# EPICS substitutions: iocBoot/ioc13idd/SIS3820_8.substitutions
# This loads the scaler record and supporting records
file "$(STD)/stdApp/Db/scaler.db"
{
pattern
{P,           S,          DTYP,           OUT,                     FREQ}
{13IDD:  scaler2,  "Asyn Scaler",  "@asyn(mcaSIS3820/1 0)",    50000000}
}

# This database provides the record for callbacks when acquisition is complete
file "$(MCA)/mcaApp/Db/SIS3820.db"
{
pattern
{P,         INP}
{13IDD:SIS1:  "@asyn(mcaSIS3820/1 0)"}
}

# This database provides the logic for multiple mca records
file "$(MCA)/mcaApp/Db/Struck8.db"
{
pattern
{P}
{13IDD:SIS1:}
}

# This loads the MCA records
file "$(MCA)/mcaApp/Db/simple_mca.db"
{
pattern
{P,           M,          DTYP,           INP, PREC, CHANS}
{13IDD:SIS1:  mca1,  "asynMCA", "@asyn(mcaSIS3820/1 0)",  3,  2048}
{13IDD:SIS1:  mca2,  "asynMCA", "@asyn(mcaSIS3820/1 1)",  3,  2048}
{13IDD:SIS1:  mca3,  "asynMCA", "@asyn(mcaSIS3820/1 2)",  3,  2048}
{13IDD:SIS1:  mca4,  "asynMCA", "@asyn(mcaSIS3820/1 3)",  3,  2048}
{13IDD:SIS1:  mca5,  "asynMCA", "@asyn(mcaSIS3820/1 4)",  3,  2048}
{13IDD:SIS1:  mca6,  "asynMCA", "@asyn(mcaSIS3820/1 5)",  3,  2048}
{13IDD:SIS1:  mca7,  "asynMCA", "@asyn(mcaSIS3820/1 6)",  3,  2048}
{13IDD:SIS1:  mca8,  "asynMCA", "@asyn(mcaSIS3820/1 7)",  3,  2048}
}
